// TIA Portal V20 export
DATA_BLOCK "DB_Analogic_Inputs"   // DB2
{ S7_Optimized_Access := 'TRUE' }
// stored: MemoryReserve 100
   VAR
      Electrical_Current_Read_Real : Real;
      Electrical_Voltage_Read_Real : Real;
      Electrical_Current_Read_UInt : UInt;
      Electrical_Voltage_Read_UInt : UInt;
   END_VAR
BEGIN
END_DATA_BLOCK
